///EL1258 | XFC, 8-channel digital input terminal with time stamp
FUNCTION_BLOCK EL1258_v0_00

END_FUNCTION_BLOCK

(* stored: Version 1.1.0.1, ProductVersion 3.1.0.25
   POU EL1258_v0_00: Id {ee9484d5-3596-4bc6-b9d7-d633d1311bfa} *)
